FUNCTION_BLOCK CustomForLights (* A simple FB with a single algorithm and REQ/CNF pair *)
  (* Standard: 61499-1 *)
  (* Version 0.0, 2006-09-03, JHC, Holobloc Inc *)
  (* Compiler header: package fb.rt.student; *)
  (* Compiler classdef: SimpleFB *)
  (* Compiler Java Sun JDK 1.5.0 *)
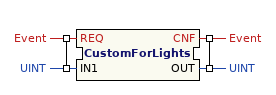
  EVENT_INPUT
    REQ WITH IN1; (* Normal Execution Request *)
  END_EVENT
  EVENT_OUTPUT
    CNF WITH OUT; (* Execution Confirmation *)
  END_EVENT
  VAR_INPUT
    IN1 : UINT;
  END_VAR
  VAR_OUTPUT
    OUT : UINT;
  END_VAR
  ALGORITHM REQ IN ST: (* Normally executed algorithm *)
IF IN1 = 0 THEN
OUT := 1;
ELSE
OUT := IN1 * 10;
END_IF;
  END_ALGORITHM
END_FUNCTION_BLOCK
